PROGRAM PRG_HMIControl
VAR
//Motor 1 Animation
rM1MotorPosition     : LREAL;  // Real Motor Actual position
rM1MotorPositionPerc : LREAL;  // Motor Actual Position Scaled 0-100
cM1MinPosition       : LREAL := 0.0; // Minimum expected Value
cM1MaxPosition       : LREAL := -320.0; // Maximum expected Value (Default Value)

//Motor 2 Animation
rM2MotorPosition     : LREAL;  // Real Motor Actual position
rM2MotorPositionPerc : LREAL;  // Motor Actual Position Scaled 0-100
cM2MinPosition       : LREAL := 0.0; // Minimum expected Value
cM2MaxPosition       : LREAL := -170.0; // Maximum expected Value (Default Value)

//Pumps Animation and status
aPumpStatus			: ARRAY[1..10] OF ST_ActuatorStatus;
fbBlinkPumpArrowFWD	: ARRAY[1..10] OF FB_Blink;
fbBlinkPumpArrowBWD	: ARRAY[1..10] OF FB_Blink;

//Headbar Machine Mode transition
fbBlinkMachineModeName 	: FB_Blink;
ePrevMode               : E_MachineMode := E_MachineMode.IMEDIATE_FAULT; 
rTrigChange             : R_TRIG;
bStateChanged           : BOOL;
tpChangePulse           : TP; // gera um pulso de PT quando IN sobe
bBlinkMode              : BOOL;

//Doors Animation
fbBlinkDoor	: ARRAY[1..6] OF FB_Blink;
fbHMIScan	: FB_Blink;

//Icons Animation
bFirstIconSet : BOOL := FALSE;

//EStops Buttons
fbBlinkEStopSide	: FB_Blink;
fbBlinkEStopFront	: FB_Blink;

//Solvent status flags
bSolventIssue : BOOL := FALSE;
ton500ms : TON;
i : INT;

//Timers for releasing interlock signals.
tonInterlockReleaseM1 : ton;
tonInterlockReleaseM2 : ton;
tonInterlockReleaseM3 : ton;

//Jars Animation
curTurns         : LREAL;
deltaTurns       : LREAL;
dMl              : LREAL;
dir              : SINT;       // -1 Fill down, +1 Fill up, 0 stopped
effDeltaMl       : LREAL;
valIdx           : INT;
displayMl        : LREAL;
segPrevEff       : LREAL;
segNowEff        : LREAL;
bRecircActive    : BOOL;
END_VAR

VAR CONSTANT
    cJarsCount              : INT   := 10;
    cJarCapacity_ml         : LREAL := 80.0;
    cDeadVolDefault_ml      : LREAL := 20.0;
    cEpsTurns               : LREAL := 1e-6;
    cRecircLowDeg           : LREAL := 4700.0;
    cRecircHighDeg          : LREAL := 4900.0;
    cRecircDisplayMin_ml    : LREAL := 20.0;   // alvo mínimo visual durante recirculação
END_VAR

VAR RETAIN
    // Integração por bomba (estado interno do jar)
    aPrevTurns       : ARRAY[1..10] OF LREAL;
    aPrevInit        : ARRAY[1..10] OF BOOL;
    aJarMl           : ARRAY[1..10] OF LREAL;

    // Segmentação por direção (fora da recirculação)
    aSegDir          : ARRAY[1..10] OF SINT;     // -1 / 0 / +1
    aSegAbsMl        : ARRAY[1..10] OF LREAL;    // mL acumulados no segmento atual (|mL|)
    aSegAbsMlPrev    : ARRAY[1..10] OF LREAL;

    // Ajustes de unidade e dead volume por bomba
    aUnitsPerTurn    : ARRAY[1..10] OF LREAL := [1(360.0),360.0,360.0,360.0,360.0,360.0,360.0,360.0,360.0,360.0]; // graus->volta
    aDeadVolCfg_ml   : ARRAY[1..10] OF LREAL := [1(cDeadVolDefault_ml),
                                                 cDeadVolDefault_ml, cDeadVolDefault_ml, cDeadVolDefault_ml, cDeadVolDefault_ml,
                                                 cDeadVolDefault_ml, cDeadVolDefault_ml, cDeadVolDefault_ml, cDeadVolDefault_ml, cDeadVolDefault_ml];

    // Exibição durante recirculação
    aRecircWasActive : ARRAY[1..10] OF BOOL;     // para detectar borda de entrada/saída
    aRecircBaseMl    : ARRAY[1..10] OF LREAL;    // patamar antes de entrar em recirculação
    aDispMl          : ARRAY[1..10] OF LREAL;    // nível exibido (pode divergir de aJarMl na recirculação)
END_VAR

//Buttons Indicators -------------------------------------------------------------------------------------------------
GVL_HMI.HMIDigOutputs.bHMIResetButton 	:= GVL_IO.gDigOutputs.bResetIndicator;
GVL_HMI.HMIDigOutputs.bHMIStartButton	:= GVL_IO.gDigOutputs.bStartIndicator;
fbBlinkEStopSide(bEnable := NOT (GVL_Safety.SafetyInputs.bEStopSideCh1 OR GVL_Safety.SafetyInputs.bEStopSideCh2), tPeriod := T#1S); //EStop Button located on side Flashing FB
fbBlinkEStopFront(bEnable := NOT (GVL_Safety.SafetyInputs.bEStopHMICh1 OR GVL_Safety.SafetyInputs.bEStopHMICh2), tPeriod := T#1S);  //EStop Button located on front Flashing FB
GVL_HMI.HMIDigOutputs.bHMIEStopSide		:= fbBlinkEStopSide.bBlink;
GVL_HMI.HMIDigOutputs.bHMIEStopFront	:= fbBlinkEStopFront.bBlink;

(* Alarm Lamp Indicator for HMI --------------------------------------------------------------------------------------- *)
GVL_HMI.HMIDigOutputs.bAlarmLampRed 	:= GVL_IO.gDigOutputs.bTowerRedLight; 	//Red Light
GVL_HMI.HMIDigOutputs.bAlarmLampAmbar 	:= GVL_IO.gDigOutputs.bTowerAmberLight; //Ambar Light
GVL_HMI.HMIDigOutputs.bAlarmLampGreen 	:= GVL_IO.gDigOutputs.bTowerGreenLight; //Green Light

(* <Controls Animation> ------------------------------------------------------------------------------------------------ *)
ACT_M1Animation();
ACT_M2Animation();

(* Head Bar Blinking *) //----------------------------------------------------------------------------------------------------
// 1) State changed?
rTrigChange(CLK := (GVL_HMI.eMachineMode <> ePrevMode));
bStateChanged := rTrigChange.Q;

// 2) Short pulse whe changed
tpChangePulse(IN := bStateChanged, PT := T#500MS);

// 3) Blinking states
bBlinkMode := (GVL_HMI.eMachineMode = E_MachineMode.SYSTEM_READY)
           OR (GVL_HMI.eMachineMode = E_MachineMode.IMEDIATE_FAULT);

// Blinking F
fbBlinkMachineModeName(bEnable := bBlinkMode, tPeriod := T#1S);

// 4) HMI Output
GVL_HMI.bMachineModeBlinking := tpChangePulse.Q OR (bBlinkMode AND fbBlinkMachineModeName.bBlink);

// 5) Update previous machine mode
ePrevMode := GVL_HMI.eMachineMode;

(* HMI Lights Control *) //-----------------------------------------------------------------------------------------------
GVL_IO.gRelayOutputs.bSampleRecoveryLight 		:= GVL_HMI.bLightsToggleButton;
GVL_IO.gRelayOutputs.bStageCollectionLeftLight 	:= GVL_HMI.bLightsToggleButton;
GVL_IO.gRelayOutputs.bStageCollectionRightLight := GVL_HMI.bLightsToggleButton;

(* <Linear Pumps Old Position> ----------------------------------------------------------------------------------------- *)
// display linear pumps old position saved on persistent memory when in Calibration Mode
IF GVL_HMI.eMachineMode = E_MachineMode.CALIBRATION THEN
	FOR i := 1 TO 10 DO
		GVL_HMI.aCalibLinearPumps[i].rOldPosition := GVL_Retain.rLinearPumpOldPosition[i];
		//pump factor
		GVL_HMI.aCalibLinearPumps[i].rPumpFactor := GVL_Motion.aPumps[1].Rotary.rActualPos;
	END_FOR
END_IF

(* <Pump Factor Showing> ----------------------------------------------------------------------------------------------- *)
(*IF GVL_HMI.eMachineMode = E_MachineMode.CALIBRATION THEN
	FOR i := 1 TO 10 DO
		GVL_HMI.aCalPumpResults[i].rPumpFactor := GVL_Motion.aPumps[i].Rotary.rPumpFactorFromCalBox;
	END_FOR
END_IF
*)

(* <Safety Controls> ----------------------------------------------------------------------------------------------------*)
ton500ms(IN := NOT ton500ms.Q, PT := T#500MS);

IF ton500ms.Q THEN ACT_IOControls(); END_IF

//Calibration Box presence
GVL_HMI.bHMICalibrationBox := GVL_IO.gDigInputs.bCalibrationBoxPresent;

//Valves Angle
GVL_HMI.HMIAnimation.aValveAngle[1]	:= GVL_Motion.aValves[1].rActualPosition / 60;
GVL_HMI.HMIAnimation.aValveAngle[2]	:= GVL_Motion.aValves[2].rActualPosition / 60;;
GVL_HMI.HMIAnimation.aValveAngle[3]	:= GVL_Motion.aValves[3].rActualPosition / 60;;
GVL_HMI.HMIAnimation.aValveAngle[4]	:= GVL_Motion.aValves[4].rActualPosition / 60;;
GVL_HMI.HMIAnimation.aValveAngle[5]	:= GVL_Motion.aValves[5].rActualPosition / 60;;

//Pumps status Running or busy
IF GVL_HMI.eMachineMode = E_MachineMode.MANUAL THEN
	FOR i := 1 TO 10 DO
		aPumpStatus[i] := GVL_Motion.aPumpsRotary[i].GetStatus();
		GVL_HMI.aManualPumpsCmd[i].bBusy := NOT GVL_Motion.aPumps[i].Rotary.iNotMoving; //aPumpStatus[i].bBusy;
	END_FOR
END_IF

//Check if there is at least one pump running
GVL_Motion.bAnyPumpRunning := FALSE;
FOR i := 1 TO 10 DO
	IF GVL_HMI.aManualPumpsCmd[i].bBusy THEN
		GVL_Motion.bAnyPumpRunning := TRUE;
		EXIT;
	END_IF
END_FOR


//Pumps Animation | Calibration Screen
IF GVL_HMI.eMachineMode = E_MachineMode.CALIBRATION THEN
	ACT_CalibrationArrows();
END_IF

//Scan period for hmi refresh
//IF GVL_HMI.eMachineMode <> E_MachineMode.CALIBRATION AND GVL_HMI.eMachineMode <> E_MachineMode.MANUAL THEN
	fbHMIScan(bEnable := GVL_HMI.bHomeScreenLoaded, tPeriod := T#500MS);
	GVL_HMI.bMachineModeScan := fbHMIScan.bBlink;
//ELSE
//	GVL_HMI.bMachineModeScan := FALSE;
//END_IF


//Doors hide/visible 
GVL_HMI.HMIAnimation.bHMIDoorOpen[1] := NOT GVL_Safety.SafetyInputs.bStageCollectLeftDoorFdbk;
GVL_HMI.HMIAnimation.bHMIDoorOpen[2] := NOT GVL_Safety.SafetyInputs.bStageCollectRightDoorFdbk;
GVL_HMI.HMIAnimation.bHMIDoorOpen[3] := NOT GVL_Safety.SafetyInputs.bSampleRecoveryDoorFdbk;
GVL_HMI.HMIAnimation.bHMIDoorOpen[4] := GVL_IO.gDigInputs.bAccessDoor4InterlockFdbk;
GVL_HMI.HMIAnimation.bHMIDoorOpen[5] := GVL_IO.gDigInputs.bAccessDoor5InterlockFdbk;
GVL_HMI.HMIAnimation.bHMIDoorOpen[6] := GVL_IO.gDigInputs.bAccessDoor6InterlockFdbk;

//Doors open blinking red alert
fbBlinkDoor[1](bEnable := NOT GVL_Safety.SafetyInputs.bStageCollectLeftDoorFdbk, tPeriod := T#1S);
GVL_HMI.HMIAnimation.bHMIDoorBlink[1] := fbBlinkDoor[1].bBlink;

fbBlinkDoor[2](bEnable := NOT GVL_Safety.SafetyInputs.bStageCollectRightDoorFdbk, tPeriod := T#1S);
GVL_HMI.HMIAnimation.bHMIDoorBlink[2] := fbBlinkDoor[2].bBlink;

fbBlinkDoor[3](bEnable := NOT GVL_Safety.SafetyInputs.bSampleRecoveryDoorFdbk, tPeriod := T#1S);
GVL_HMI.HMIAnimation.bHMIDoorBlink[3] := fbBlinkDoor[3].bBlink;

fbBlinkDoor[4](bEnable := GVL_IO.gDigInputs.bAccessDoor4InterlockFdbk, tPeriod := T#1S);
GVL_HMI.HMIAnimation.bHMIDoorBlink[4] := fbBlinkDoor[4].bBlink;

fbBlinkDoor[5](bEnable := GVL_IO.gDigInputs.bAccessDoor5InterlockFdbk, tPeriod := T#1S);
GVL_HMI.HMIAnimation.bHMIDoorBlink[5] := fbBlinkDoor[5].bBlink;

fbBlinkDoor[6](bEnable := GVL_IO.gDigInputs.bAccessDoor6InterlockFdbk, tPeriod := T#1S);
GVL_HMI.HMIAnimation.bHMIDoorBlink[6] := fbBlinkDoor[6].bBlink;


(* <\Controls Animation> *********************************************************************************************** *)

(* <Icons Animation> *************************************************************************************************** *)
IF NOT bFirstIconSet THEN
	GVL_HMI.HMIAnimation.eIconStateSafety   := E_IconState.Waiting;
	GVL_HMI.HMIAnimation.eIconStateAirFlow  := E_IconState.Waiting;
	GVL_HMI.HMIAnimation.eIconStateHardware := E_IconState.Waiting;
	GVL_HMI.HMIAnimation.eIconStateLeakTest := E_IconState.Waiting;
	GVL_HMI.HMIAnimation.eIconStateRecovery := E_IconState.Waiting;
	GVL_HMI.HMIAnimation.eIconStateWashing  := E_IconState.Waiting;
	GVL_HMI.HMIAnimation.eIconStateDry 		:= E_IconState.Waiting;
	bFirstIconSet := TRUE;
END_IF

IF GVL_HMI.eMachineMode = E_MachineMode.IMEDIATE_FAULT THEN
	GVL_HMI.HMIAnimation.eIconStateSafety   := E_IconState.Waiting;
	GVL_HMI.HMIAnimation.eIconStateAirFlow  := E_IconState.Waiting;
	GVL_HMI.HMIAnimation.eIconStateHardware := E_IconState.Waiting;
	GVL_HMI.HMIAnimation.eIconStateLeakTest := E_IconState.Waiting;
	GVL_HMI.HMIAnimation.eIconStateRecovery := E_IconState.Waiting;
	GVL_HMI.HMIAnimation.eIconStateWashing  := E_IconState.Waiting;
	GVL_HMI.HMIAnimation.eIconStateDry 	    := E_IconState.Waiting;
ELSE
	GVL_HMI.HMIAnimation.eIconStateSafety := E_IconState.Completed;
END_IF

IF GVL_HMI.eMachineMode = E_MachineMode.STOPPED THEN
	GVL_HMI.HMIAnimation.eIconStateSafety   := E_IconState.Waiting;
	GVL_HMI.HMIAnimation.eIconStateAirFlow  := E_IconState.Waiting;
	GVL_HMI.HMIAnimation.eIconStateHardware := E_IconState.Waiting;
	GVL_HMI.HMIAnimation.eIconStateLeakTest := E_IconState.Waiting;
	GVL_HMI.HMIAnimation.eIconStateRecovery := E_IconState.Waiting;
	GVL_HMI.HMIAnimation.eIconStateWashing  := E_IconState.Waiting;
	GVL_HMI.HMIAnimation.eIconStateDry 	    := E_IconState.Waiting;
END_IF

(* <\Icons Animation> *************************************************************************************************** *)

(* <Machine Settings> ************************************************************************************************** *)
IF GVL_HMI.bSaveParametersBt THEN // Save Settings button from HMI
	GVL_Settings.stMachineParam	 		:= GVL_HMI.HMIParameters; 		 // Motion Settings
	GVL_Settings.stCalibParameters 		:= GVL_HMI.stHMICalibParameters; // Calibration Settings
	GVL_Settings.stPumpParameters 		:= GVL_HMI.stHMIPumpParameters;	 // Pump Settings
	GVL_Settings.stLeakTestParameters 	:= GVL_HMI.stLeakTestParameters; // Leak Test Settings
	GVL_HMI.bSaveParametersBt 	:= FALSE;
	GVL_HMI.bSaveParametersDone := TRUE;
END_IF

IF GVL_HMI.bReloadHMIParameters OR (GVL_HMI.eMachineMode = E_MachineMode.CALIBRATION) THEN
	GVL_HMI.HMIParameters := GVL_Settings.stMachineParam;				 // Motion Settings
	GVL_HMI.stHMICalibParameters := GVL_Settings.stCalibParameters; 	 // Calibration Settings
	GVL_HMI.stHMIPumpParameters  := GVL_Settings.stPumpParameters; 		 // Pump Settings
	GVL_HMI.stLeakTestParameters := GVL_Settings.stLeakTestParameters; 	 // Leak Test Settings
	GVL_HMI.bReloadHMIParameters := FALSE;
END_IF
(* <\Machine Settings> ************************************************************************************************** *)

(* <HMI Alerts> ********************************************************************************************************* *)

//Auto Cycle Incoherence [when there is something missing to start the auto cycle] 
GVL_HMI.bIncoherenceDetected := (NOT GVL_Recipe.bIsThereRecipeActivated) OR (NOT GVL_IO.gDigInputs.bThroatJigPresent) OR (NOT GVL_IO.bVialRackPresent) OR bSolventIssue;

bSolventIssue := GVL_Alarms.aSolventLowLevel[1] OR GVL_Alarms.aSolventLowLevel[2] OR GVL_Alarms.aSolventLowLevel[3] OR GVL_Alarms.aSolventLowLevel[4] OR GVL_Alarms.bWasteHighLevel;

IF GVL_HMI.HMIAnimation.rWasteLevel	> 70 THEN
	GVL_Alarms.bWasteHighLevel := TRUE;
ELSE
	GVL_Alarms.bWasteHighLevel := FALSE;
END_IF

IF GVL_Recipe.bIsThereRecipeActivated THEN
	//Checking solvent levels of Rinse 1 Solvent
	CASE GVL_Recipe.stActiveRecipe.stSolventsTimes.aSolventN[1] OF
	1:
		IF GVL_HMI.HMIAnimation.aSolventLevel[1] < 30 THEN
			GVL_Alarms.aSolventLowLevel[1] := TRUE;
		ELSE
			GVL_Alarms.aSolventLowLevel[1] := FALSE;
		END_IF
	2:
		IF GVL_HMI.HMIAnimation.aSolventLevel[2] < 30 THEN
			GVL_Alarms.aSolventLowLevel[2] := TRUE;
		ELSE
			GVL_Alarms.aSolventLowLevel[2] := FALSE;
		END_IF

	3:
		IF GVL_HMI.HMIAnimation.aSolventLevel[3] < 30 THEN
			GVL_Alarms.aSolventLowLevel[3] := TRUE;
		ELSE
			GVL_Alarms.aSolventLowLevel[3] := FALSE;
		END_IF
	4:
		IF GVL_HMI.HMIAnimation.aSolventLevel[4] < 30 THEN
			GVL_Alarms.aSolventLowLevel[4] := TRUE;
		ELSE
			GVL_Alarms.aSolventLowLevel[4] := FALSE;
		END_IF
	END_CASE 
	
	//Checking solvent levels of Rinse 2 Solvent
	CASE GVL_Recipe.stActiveRecipe.stSolventsTimes.aSolventN[2] OF
	1:
		IF GVL_HMI.HMIAnimation.aSolventLevel[1] < 30 THEN
			GVL_Alarms.aSolventLowLevel[1] := TRUE;
		ELSE
			GVL_Alarms.aSolventLowLevel[1] := FALSE;
		END_IF
	2:
		IF GVL_HMI.HMIAnimation.aSolventLevel[2] < 30 THEN
			GVL_Alarms.aSolventLowLevel[2] := TRUE;
		ELSE
			GVL_Alarms.aSolventLowLevel[2] := FALSE;
		END_IF

	3:
		IF GVL_HMI.HMIAnimation.aSolventLevel[3] < 30 THEN
			GVL_Alarms.aSolventLowLevel[3] := TRUE;
		ELSE
			GVL_Alarms.aSolventLowLevel[3] := FALSE;
		END_IF
	4:
		IF GVL_HMI.HMIAnimation.aSolventLevel[4] < 30 THEN
			GVL_Alarms.aSolventLowLevel[4] := TRUE;
		ELSE
			GVL_Alarms.aSolventLowLevel[4] := FALSE;
		END_IF
	END_CASE 
END_IF

//-------------------------------------------------

IF GVL_Recipe.bIsThereRecipeActivated THEN
	GVL_HMI.sActivatedRecipeHomeNaming := concat(GVL_Recipe.stActiveRecipe.stInfo.sMethodName,concat(' | Created by ', concat(GVL_Recipe.stActiveRecipe.stInfo.sCreatedBy,concat(' on ', DATE_TO_STRING(GVL_Recipe.stActiveRecipe.stInfo.dCreationDate)))));
ELSE
	GVL_HMI.sActivatedRecipeHomeNaming := 'There is no Recipe Activated';
END_IF

(* <\HMI Alerts> ******************************************************************************************************* *)
(* Motors Interlock *) // Releasing alarm trigger after 2 seconds.
IF GVL_HMI.bM1MoveNotAllowedTrigger THEN
	tonInterlockReleaseM1(In := TRUE, PT := T#2S);
ELSE
	tonInterlockReleaseM1(In := FALSE, PT := T#2S);
END_IF

IF GVL_HMI.bM2MoveNotAllowedTrigger THEN
	tonInterlockReleaseM2(In := TRUE, PT := T#2S);
ELSE
	tonInterlockReleaseM2(In := FALSE, PT := T#2S);
END_IF

IF GVL_HMI.bM3MoveNotAllowedTrigger THEN
	tonInterlockReleaseM3(In := TRUE, PT := T#2S);
ELSE
	tonInterlockReleaseM3(In := FALSE, PT := T#2S);
END_IF

IF tonInterlockReleaseM1.Q THEN
	GVL_HMI.bM1MoveNotAllowedTrigger := FALSE;
END_IF

IF tonInterlockReleaseM2.Q THEN
	GVL_HMI.bM2MoveNotAllowedTrigger := FALSE;
END_IF

IF tonInterlockReleaseM3.Q THEN
	GVL_HMI.bM3MoveNotAllowedTrigger := FALSE;
END_IF

(* <TEMP ******************************************************************************************************* *)
IF GVL_HMI.bResetM1MotorBt THEN
	GVL_HMI.bResetM1MotorBt := NOT GVL_Motion.aMotors[1].Reset();
END_IF

ACTION ACT_CalibrationArrows:
(* Pumps arrow animation *)
//Get pump Status
FOR i := 1 TO 10 DO
	aPumpStatus[i] := GVL_Motion.aPumpsRotary[i].GetStatus();
END_FOR

//Blink aPumpMovingFwd[i] if moving forward
FOR i := 1 TO 10 DO
	fbBlinkPumpArrowFWD[i]( bEnable := aPumpStatus[i].bMovingFwd, tPeriod := T#500MS );
	GVL_HMI.HMIAnimation.aPumpingArrowFwd[i] := fbBlinkPumpArrowFWD[i].bBlink;
END_FOR

//Blink aPumpMovingBwd[i] if moving backwards
FOR i := 1 TO 10 DO
	fbBlinkPumpArrowBWD[i]( bEnable := aPumpStatus[i].bMovingBck, tPeriod := T#500MS );
	GVL_HMI.HMIAnimation.aPumpingArrowBwd[i] := fbBlinkPumpArrowBWD[i].bBlink;
END_FOR
END_ACTION

ACTION ACT_IOControls:

(* <EL6910 Terminal 3> -------------------------------------------------------------------------------------------------------------*)
GVL_IO.stEL6910.qSafetyRun 			:= GVL_Safety.bSafetyRun;
GVL_IO.stEL6910.qSafetyErrorAck 	:= GVL_Safety.bSafetyErrorAck;
GVL_IO.stEL6910.qSafetyAirPresureOK := GVL_Safety.SafetyOutputs.bAirPressureOK;
GVL_IO.stEL6910.iSafetyOK 			:= GVL_Safety.bSafetyEnable;
GVL_IO.stEL6910.qLockDoorsCommand	:= GVL_Safety.bDoorLockCommand;
GVL_IO.stEL6910.iBypassDoor3Command := GVL_Safety.bDoor3BypassAccepted;


(* <EL1918 Terminal 4> -------------------------------------------------------------------------------------------------------------*)
GVL_HMI.aIOTerm04[1] := GVL_Safety.SafetyInputs.bEStopHMICh1;
GVL_HMI.aIOTerm04[2] := GVL_Safety.SafetyInputs.bEStopHMICh2;
GVL_HMI.aIOTerm04[3] := GVL_Safety.SafetyInputs.bEStopSideCh1;
GVL_HMI.aIOTerm04[4] := GVL_Safety.SafetyInputs.bEStopSideCh2;
GVL_HMI.aIOTerm04[5] := GVL_Safety.SafetyInputs.bMachineReset;
GVL_HMI.aIOTerm04[6] := GVL_Safety.SafetyInputs.bStageCollectLeftDoorCh1;
GVL_HMI.aIOTerm04[7] := GVL_Safety.SafetyInputs.bStageCollectLeftDoorCh2;
GVL_HMI.aIOTerm04[8] := GVL_Safety.SafetyInputs.bStageCollectLeftDoorFdbk;

(* <EL1918 Terminal 5> -------------------------------------------------------------------------------------------------------------*)
GVL_HMI.aIOTerm05[1] := GVL_Safety.SafetyInputs.bStageCollectRightDoorCh1;
GVL_HMI.aIOTerm05[2] := GVL_Safety.SafetyInputs.bStageCollectRightDoorCh2;
GVL_HMI.aIOTerm05[3] := GVL_Safety.SafetyInputs.bStageCollectRightDoorFdbk;
GVL_HMI.aIOTerm05[4] := GVL_Safety.SafetyInputs.bSampleRecoveryDoorCh1;
GVL_HMI.aIOTerm05[5] := GVL_Safety.SafetyInputs.bSampleRecoveryDoorCh2;
GVL_HMI.aIOTerm05[6] := GVL_Safety.SafetyInputs.bSampleRecoveryDoorFdbk;
GVL_HMI.aIOTerm05[7] := FALSE;
GVL_HMI.aIOTerm05[8] := FALSE;

(* <EL1918 Terminal 6> -------------------------------------------------------------------------------------------------------------*)
GVL_HMI.aIOTerm06[1] := NOT GVL_Safety.SafetyInputs.bFestoMS6ValveFdbk;
GVL_HMI.aIOTerm06[2] := GVL_Safety.SafetyInputs.bFestoMS6DumpValveFdbk;
GVL_HMI.aIOTerm06[3] := NOT GVL_Safety.SafetyInputs.bD4AccessDoorIntlckOSSD1;
GVL_HMI.aIOTerm06[4] := NOT GVL_Safety.SafetyInputs.bD4AccessDoorIntlckOSSD2;
GVL_HMI.aIOTerm06[5] := NOT GVL_Safety.SafetyInputs.bD5AccessDoorIntlckOSSD1;
GVL_HMI.aIOTerm06[6] := NOT GVL_Safety.SafetyInputs.bD5AccessDoorIntlckOSSD2;
GVL_HMI.aIOTerm06[7] := NOT GVL_Safety.SafetyInputs.bD6AccessDoorIntlckOSSD1;
GVL_HMI.aIOTerm06[8] := NOT GVL_Safety.SafetyInputs.bD6AccessDoorIntlckOSSD2;

(* <EL2904 Terminal 7> -------------------------------------------------------------------------------------------------------------*)
GVL_HMI.aIOTerm07[1] := GVL_Safety.aEL2904_T07[1];
GVL_HMI.aIOTerm07[2] := GVL_Safety.aEL2904_T07[2];
GVL_HMI.aIOTerm07[3] := GVL_Safety.aEL2904_T07[3];
GVL_HMI.aIOTerm07[4] := GVL_Safety.aEL2904_T07[4];

(* <EL2904 Terminal 8> -------------------------------------------------------------------------------------------------------------*)
GVL_HMI.aIOTerm08[1] := GVL_Safety.aEL2904_T08[1];
GVL_HMI.aIOTerm08[2] := GVL_Safety.aEL2904_T08[2];
GVL_HMI.aIOTerm08[3] := GVL_Safety.aEL2904_T08[3];
GVL_HMI.aIOTerm08[4] := GVL_Safety.aEL2904_T08[4];

(* <EL1809 Terminal 9> -------------------------------------------------------------------------------------------------------------*)
GVL_HMI.aIOTerm09[1] := GVL_IO.gDigInputs.bStartButton;
GVL_HMI.aIOTerm09[2] := GVL_IO.gDigInputs.bStopButton;
GVL_HMI.aIOTerm09[3] := GVL_IO.gDigInputs.b24VPowerSupplyOK;
GVL_HMI.aIOTerm09[4] := GVL_IO.gDigInputs.b24VPowerSupplyOKBck;
GVL_HMI.aIOTerm09[5] := GVL_IO.gDigInputs.b48VPowerSupplyOK;
GVL_HMI.aIOTerm09[6] := GVL_IO.gDigInputs.bStageCollection_Home;
GVL_HMI.aIOTerm09[7] := GVL_IO.gDigInputs.bSampleRecovery_Vertical_Home;
GVL_HMI.aIOTerm09[8] := GVL_IO.gDigInputs.bSampleRecovery_Horizontal_Home;
GVL_HMI.aIOTerm09[9] := GVL_IO.gDigInputs.bWasteOverflowSensor;
GVL_HMI.aIOTerm09[10] := GVL_IO.gDigInputs.bUPSReady;
GVL_HMI.aIOTerm09[11] := GVL_IO.gDigInputs.bUPSReplaceBattery;
GVL_HMI.aIOTerm09[12] := GVL_IO.gDigInputs.b48VPowerSupplyOKBck;
GVL_HMI.aIOTerm09[13] := GVL_IO.gDigInputs.bCalibrationBoxPresent;
GVL_HMI.aIOTerm09[14] := GVL_IO.gDigInputs.bThroatJigPresent;
GVL_HMI.aIOTerm09[15] := FALSE;
GVL_HMI.aIOTerm09[16] := FALSE;

(* <EL2809 Terminal 10> -------------------------------------------------------------------------------------------------------------*)
GVL_HMI.aIOTerm10[1] := GVL_IO.gDigOutputs.bStartIndicator;
GVL_HMI.aIOTerm10[2] := GVL_IO.gDigOutputs.bResetIndicator;
GVL_HMI.aIOTerm10[3] := GVL_IO.gDigOutputs.bTowerRedLight;
GVL_HMI.aIOTerm10[4] := GVL_IO.gDigOutputs.bTowerAmberLight;
GVL_HMI.aIOTerm10[5] := GVL_IO.gDigOutputs.bTowerGreenLight;
GVL_HMI.aIOTerm10[6] := GVL_IO.gDigOutputs.bTowerBuzzer;
GVL_HMI.aIOTerm10[7] := GVL_IO.gDigOutputs.bSolenoidValveB;
GVL_HMI.aIOTerm10[8] := GVL_IO.gDigOutputs.bSolenoidValveA;
GVL_HMI.aIOTerm10[9] := GVL_IO.gDigOutputs.bSolenoidValveC;
GVL_HMI.aIOTerm10[10] := FALSE;
GVL_HMI.aIOTerm10[11] := FALSE;
GVL_HMI.aIOTerm10[12] := FALSE;
GVL_HMI.aIOTerm10[13] := FALSE;
GVL_HMI.aIOTerm10[14] := FALSE;
GVL_HMI.aIOTerm10[15] := FALSE;
GVL_HMI.aIOTerm10[16] := FALSE;

(* <EL2624 Terminal 11> -------------------------------------------------------------------------------------------------------------*)
GVL_HMI.aIOTerm11[1] := GVL_IO.gRelayOutputs.bStageCollectionLeftLight;
GVL_HMI.aIOTerm11[2] := GVL_IO.gRelayOutputs.bSampleRecoveryLight;
GVL_HMI.aIOTerm11[3] := GVL_IO.gRelayOutputs.bStageCollectionRightLight;
GVL_HMI.aIOTerm11[4] := FALSE;

(* <EL9410 Terminal 12> -------------------------------------------------------------------------------------------------------------*)
GVL_HMI.aIOTerm12[1] := GVL_IO.bEL9410UPStatus;
GVL_HMI.aIOTerm12[2] := GVL_IO.bEL9410USStatus;

(* <EL3058 Terminal 13> -------------------------------------------------------------------------------------------------------------*)
GVL_HMI.aIOTerm13[1] := GVL_IO.gAnalogInputs.rMainPressureSupplyInput;
GVL_HMI.aIOTerm13[2] := GVL_IO.gAnalogInputs.rLeakTestPressureSensor;
GVL_HMI.aIOTerm13[3] := GVL_IO.gAnalogInputs.rPressureRegulatorInput;
GVL_HMI.aIOTerm13[3] := 0.0;

(* <EL9576 Terminal 14> -------------------------------------------------------------------------------------------------------------*)
GVL_HMI.aIOTerm14[1] := GVL_IO.bEL9576T14Overtemp;
GVL_HMI.aIOTerm14[2] := GVL_IO.bEL9576T14I2TError;
GVL_HMI.aIOTerm14[3] := GVL_IO.bEL9576T14I2TWarning;
GVL_HMI.aIOTerm14[4] := GVL_IO.bEL9576T14OverVoltage;
GVL_HMI.aIOTerm14[5] := GVL_IO.bEL9576T14UnderVoltage;
GVL_HMI.aIOTerm14[6] := GVL_IO.bEL9576T14ChopperOn;
GVL_HMI.aIOTerm14[7] := GVL_IO.bEL9576T14OverCurrent;
GVL_HMI.iIOTerm14DCIn := GVL_IO.bEL9576T14DCLinkVoltage;

(* <EL7211 Terminal 15> -------------------------------------------------------------------------------------------------------------*)
GVL_HMI.aIOTerm15[1] := GVL_Motion.M2Motor.iOperational;
GVL_HMI.aIOTerm15[2] := GVL_Motion.M2Motor.iHomed;
GVL_HMI.aIOTerm15[3] := GVL_Motion.M2Motor.iError;
GVL_HMI.aIOTerm15Values[1] := LINT_TO_LREAL(TRUNC(GVL_Motion.M2Motor.rActualPosition*1000)) / 1000.0;
GVL_HMI.aIOTerm15Values[2] := LINT_TO_LREAL(TRUNC(GVL_Motion.M2Motor.rActualVel*1000)) / 1000.0;
GVL_HMI.aIOTerm15Values[3] := LINT_TO_LREAL(TRUNC(GVL_Motion.M2Motor.rActualTorque*1000)) / 1000.0;
GVL_HMI.iIOTerm15ErrorCode := GVL_Motion.M2Motor.nErrorCode;

(* <EL7211 Terminal 16> -------------------------------------------------------------------------------------------------------------*)
GVL_HMI.aIOTerm16[1] := GVL_Motion.M3Motor.iOperational;
GVL_HMI.aIOTerm16[2] := GVL_Motion.M3Motor.iHomed;
GVL_HMI.aIOTerm16[3] := GVL_Motion.M3Motor.iError;
GVL_HMI.aIOTerm16Values[1] := LINT_TO_LREAL(TRUNC(GVL_Motion.M3Motor.rActualPosition*1000)) / 1000.0;
GVL_HMI.aIOTerm16Values[2] := LINT_TO_LREAL(TRUNC(GVL_Motion.M3Motor.rActualVel*1000)) / 1000.0;
GVL_HMI.aIOTerm16Values[3] := LINT_TO_LREAL(TRUNC(GVL_Motion.M3Motor.rActualTorque*1000)) / 1000.0;
GVL_HMI.iIOTerm16ErrorCode := GVL_Motion.M3Motor.nErrorCode;

(* <EL3022 Terminal 17> -------------------------------------------------------------------------------------------------------------*)
GVL_HMI.aIOTerm17[1] := GVL_IO.bEL3022ChAUnderRange;
GVL_HMI.aIOTerm17[2] := GVL_IO.bEL3022ChAOverRange;
GVL_HMI.aIOTerm17[3] := GVL_IO.bEL3022ChAError;
GVL_HMI.aIOTerm17[4] := GVL_IO.bEL3022ChBUnderRange;
GVL_HMI.aIOTerm17[5] := GVL_IO.bEL3022ChBOverRange;
GVL_HMI.aIOTerm17[6] := GVL_IO.bEL3022ChBError;
GVL_HMI.aIOTerm17Values[1] := 0.0;
GVL_HMI.aIOTerm17Values[2] := 0.0;

(* <EL1809 Terminal 18> -------------------------------------------------------------------------------------------------------------*)
GVL_HMI.aIOTerm18[1] := NOT GVL_IO.gDigInputs.bAccessDoor4InterlockFdbk;
GVL_HMI.aIOTerm18[2] := NOT GVL_IO.gDigInputs.bAccessDoor5InterlockFdbk;
GVL_HMI.aIOTerm18[3] := NOT GVL_IO.gDigInputs.bAccessDoor6InterlockFdbk;
GVL_HMI.aIOTerm18[4] := FALSE;
GVL_HMI.aIOTerm18[5] := FALSE;
GVL_HMI.aIOTerm18[6] := FALSE;
GVL_HMI.aIOTerm18[7] := FALSE;
GVL_HMI.aIOTerm18[8] := FALSE;
GVL_HMI.aIOTerm18[9] := FALSE;
GVL_HMI.aIOTerm18[10] := FALSE;
GVL_HMI.aIOTerm18[11] := FALSE;
GVL_HMI.aIOTerm18[12] := FALSE;
GVL_HMI.aIOTerm18[13] := FALSE;
GVL_HMI.aIOTerm18[14] := FALSE;
GVL_HMI.aIOTerm18[15] := FALSE;
GVL_HMI.aIOTerm18[16] := FALSE;

(* <EL2904 Terminal 19> -------------------------------------------------------------------------------------------------------------*)
GVL_HMI.aIOTerm19[1] := GVL_Safety.aEL2904_T19[1];
GVL_HMI.aIOTerm19[2] := GVL_Safety.aEL2904_T19[2];
GVL_HMI.aIOTerm19[3] := GVL_Safety.aEL2904_T19[3];
GVL_HMI.aIOTerm19[4] := GVL_Safety.aEL2904_T19[4];

(* <EL7062 Terminal 23> -------------------------------------------------------------------------------------------------------------*)
GVL_HMI.stIOTerm23.bAxisOperational[1] 	:= GVL_Motion.aPumps[1].Linear.iOperational;
GVL_HMI.stIOTerm23.rActualPosition[1] 	:= GVL_Motion.aPumps[1].Linear.rActualPos;
GVL_HMI.stIOTerm23.rActualVelocity[1] 	:= GVL_Motion.aPumps[1].Linear.rActualVel;
GVL_HMI.stIOTerm23.rActualTorque[1] 	:= GVL_Motion.aPumps[1].Linear.rActualTorque;
GVL_HMI.stIOTerm23.bAxisHomed[1] 		:= GVL_Motion.aPumps[1].Linear.iHomed;
GVL_HMI.stIOTerm23.bAxisError[1] 		:= GVL_Motion.aPumps[1].Linear.iError;
GVL_HMI.stIOTerm23.nErrorCode[1] 		:= GVL_Motion.aPumps[1].Linear.nErrorCode;
GVL_HMI.stIOTerm23.bAxisOperational[2] 	:= GVL_Motion.aPumps[1].Rotary.iOperational;
GVL_HMI.stIOTerm23.rActualPosition[2] 	:= GVL_Motion.aPumps[1].Rotary.rActualPos;
GVL_HMI.stIOTerm23.rActualVelocity[2] 	:= GVL_Motion.aPumps[1].Rotary.rActualVel;
GVL_HMI.stIOTerm23.rActualTorque[2] 	:= GVL_Motion.aPumps[1].Rotary.rActualTorque;
GVL_HMI.stIOTerm23.bAxisHomed[2] 		:= GVL_Motion.aPumps[1].Rotary.iHomed;
GVL_HMI.stIOTerm23.bAxisError[2] 		:= GVL_Motion.aPumps[1].Rotary.iError;
GVL_HMI.stIOTerm23.nErrorCode[2] 		:= GVL_Motion.aPumps[1].Rotary.nErrorCode;

(* <EL7062 Terminal 24> -------------------------------------------------------------------------------------------------------------*)
GVL_HMI.stIOTerm24.bAxisOperational[1] 	:= GVL_Motion.aPumps[2].Linear.iOperational;
GVL_HMI.stIOTerm24.rActualPosition[1] 	:= GVL_Motion.aPumps[2].Linear.rActualPos;
GVL_HMI.stIOTerm24.rActualVelocity[1] 	:= GVL_Motion.aPumps[2].Linear.rActualVel;
GVL_HMI.stIOTerm24.rActualTorque[1] 	:= GVL_Motion.aPumps[2].Linear.rActualTorque;
GVL_HMI.stIOTerm24.bAxisHomed[1] 		:= GVL_Motion.aPumps[2].Linear.iHomed;
GVL_HMI.stIOTerm24.bAxisError[1] 		:= GVL_Motion.aPumps[2].Linear.iError;
GVL_HMI.stIOTerm24.nErrorCode[1] 		:= GVL_Motion.aPumps[2].Linear.nErrorCode;
GVL_HMI.stIOTerm24.bAxisOperational[2] 	:= GVL_Motion.aPumps[2].Rotary.iOperational;
GVL_HMI.stIOTerm24.rActualPosition[2] 	:= GVL_Motion.aPumps[2].Rotary.rActualPos;
GVL_HMI.stIOTerm24.rActualVelocity[2] 	:= GVL_Motion.aPumps[2].Rotary.rActualVel;
GVL_HMI.stIOTerm24.rActualTorque[2] 	:= GVL_Motion.aPumps[2].Rotary.rActualTorque;
GVL_HMI.stIOTerm24.bAxisHomed[2] 		:= GVL_Motion.aPumps[2].Rotary.iHomed;
GVL_HMI.stIOTerm24.bAxisError[2] 		:= GVL_Motion.aPumps[2].Rotary.iError;
GVL_HMI.stIOTerm24.nErrorCode[2] 		:= GVL_Motion.aPumps[2].Rotary.nErrorCode;

(* <EL7062 Terminal 25> -------------------------------------------------------------------------------------------------------------*)
GVL_HMI.stIOTerm25.bAxisOperational[1] 	:= GVL_Motion.aPumps[3].Linear.iOperational;
GVL_HMI.stIOTerm25.rActualPosition[1] 	:= GVL_Motion.aPumps[3].Linear.rActualPos;
GVL_HMI.stIOTerm25.rActualVelocity[1] 	:= GVL_Motion.aPumps[3].Linear.rActualVel;
GVL_HMI.stIOTerm25.rActualTorque[1] 	:= GVL_Motion.aPumps[3].Linear.rActualTorque;
GVL_HMI.stIOTerm25.bAxisHomed[1] 		:= GVL_Motion.aPumps[3].Linear.iHomed;
GVL_HMI.stIOTerm25.bAxisError[1] 		:= GVL_Motion.aPumps[3].Linear.iError;
GVL_HMI.stIOTerm25.nErrorCode[1] 		:= GVL_Motion.aPumps[3].Linear.nErrorCode;
GVL_HMI.stIOTerm25.bAxisOperational[2] 	:= GVL_Motion.aPumps[3].Rotary.iOperational;
GVL_HMI.stIOTerm25.rActualPosition[2] 	:= GVL_Motion.aPumps[3].Rotary.rActualPos;
GVL_HMI.stIOTerm25.rActualVelocity[2] 	:= GVL_Motion.aPumps[3].Rotary.rActualVel;
GVL_HMI.stIOTerm25.rActualTorque[2] 	:= GVL_Motion.aPumps[3].Rotary.rActualTorque;
GVL_HMI.stIOTerm25.bAxisHomed[2] 		:= GVL_Motion.aPumps[3].Rotary.iHomed;
GVL_HMI.stIOTerm25.bAxisError[2] 		:= GVL_Motion.aPumps[3].Rotary.iError;
GVL_HMI.stIOTerm25.nErrorCode[2] 		:= GVL_Motion.aPumps[3].Rotary.nErrorCode;

(* <EL7062 Terminal 26> -------------------------------------------------------------------------------------------------------------*)
GVL_HMI.stIOTerm26.bAxisOperational[1] 	:= GVL_Motion.aPumps[4].Linear.iOperational;
GVL_HMI.stIOTerm26.rActualPosition[1] 	:= GVL_Motion.aPumps[4].Linear.rActualPos;
GVL_HMI.stIOTerm26.rActualVelocity[1] 	:= GVL_Motion.aPumps[4].Linear.rActualVel;
GVL_HMI.stIOTerm26.rActualTorque[1] 	:= GVL_Motion.aPumps[4].Linear.rActualTorque;
GVL_HMI.stIOTerm26.bAxisHomed[1] 		:= GVL_Motion.aPumps[4].Linear.iHomed;
GVL_HMI.stIOTerm26.bAxisError[1] 		:= GVL_Motion.aPumps[4].Linear.iError;
GVL_HMI.stIOTerm26.nErrorCode[1] 		:= GVL_Motion.aPumps[4].Linear.nErrorCode;
GVL_HMI.stIOTerm26.bAxisOperational[2] 	:= GVL_Motion.aPumps[4].Rotary.iOperational;
GVL_HMI.stIOTerm26.rActualPosition[2] 	:= GVL_Motion.aPumps[4].Rotary.rActualPos;
GVL_HMI.stIOTerm26.rActualVelocity[2] 	:= GVL_Motion.aPumps[4].Rotary.rActualVel;
GVL_HMI.stIOTerm26.rActualTorque[2] 	:= GVL_Motion.aPumps[4].Rotary.rActualTorque;
GVL_HMI.stIOTerm26.bAxisHomed[2] 		:= GVL_Motion.aPumps[4].Rotary.iHomed;
GVL_HMI.stIOTerm26.bAxisError[2] 		:= GVL_Motion.aPumps[4].Rotary.iError;
GVL_HMI.stIOTerm26.nErrorCode[2] 		:= GVL_Motion.aPumps[4].Rotary.nErrorCode;

(* <EL7062 Terminal 27> -------------------------------------------------------------------------------------------------------------*)
GVL_HMI.stIOTerm27.bAxisOperational[1] 	:= GVL_Motion.aPumps[5].Linear.iOperational;
GVL_HMI.stIOTerm27.rActualPosition[1] 	:= GVL_Motion.aPumps[5].Linear.rActualPos;
GVL_HMI.stIOTerm27.rActualVelocity[1] 	:= GVL_Motion.aPumps[5].Linear.rActualVel;
GVL_HMI.stIOTerm27.rActualTorque[1] 	:= GVL_Motion.aPumps[5].Linear.rActualTorque;
GVL_HMI.stIOTerm27.bAxisHomed[1] 		:= GVL_Motion.aPumps[5].Linear.iHomed;
GVL_HMI.stIOTerm27.bAxisError[1] 		:= GVL_Motion.aPumps[5].Linear.iError;
GVL_HMI.stIOTerm27.nErrorCode[1] 		:= GVL_Motion.aPumps[5].Linear.nErrorCode;
GVL_HMI.stIOTerm27.bAxisOperational[2] 	:= GVL_Motion.aPumps[5].Rotary.iOperational;
GVL_HMI.stIOTerm27.rActualPosition[2] 	:= GVL_Motion.aPumps[5].Rotary.rActualPos;
GVL_HMI.stIOTerm27.rActualVelocity[2] 	:= GVL_Motion.aPumps[5].Rotary.rActualVel;
GVL_HMI.stIOTerm27.rActualTorque[2] 	:= GVL_Motion.aPumps[5].Rotary.rActualTorque;
GVL_HMI.stIOTerm27.bAxisHomed[2] 		:= GVL_Motion.aPumps[5].Rotary.iHomed;
GVL_HMI.stIOTerm27.bAxisError[2] 		:= GVL_Motion.aPumps[5].Rotary.iError;
GVL_HMI.stIOTerm27.nErrorCode[2] 		:= GVL_Motion.aPumps[5].Rotary.nErrorCode;

(* <EL7062 Terminal 28> -------------------------------------------------------------------------------------------------------------*)
GVL_HMI.stIOTerm28.bAxisOperational[1] 	:= GVL_Motion.aPumps[6].Linear.iOperational;
GVL_HMI.stIOTerm28.rActualPosition[1] 	:= GVL_Motion.aPumps[6].Linear.rActualPos;
GVL_HMI.stIOTerm28.rActualVelocity[1] 	:= GVL_Motion.aPumps[6].Linear.rActualVel;
GVL_HMI.stIOTerm28.rActualTorque[1] 	:= GVL_Motion.aPumps[6].Linear.rActualTorque;
GVL_HMI.stIOTerm28.bAxisHomed[1] 		:= GVL_Motion.aPumps[6].Linear.iHomed;
GVL_HMI.stIOTerm28.bAxisError[1] 		:= GVL_Motion.aPumps[6].Linear.iError;
GVL_HMI.stIOTerm28.nErrorCode[1] 		:= GVL_Motion.aPumps[6].Linear.nErrorCode;
GVL_HMI.stIOTerm28.bAxisOperational[2] 	:= GVL_Motion.aPumps[6].Rotary.iOperational;
GVL_HMI.stIOTerm28.rActualPosition[2] 	:= GVL_Motion.aPumps[6].Rotary.rActualPos;
GVL_HMI.stIOTerm28.rActualVelocity[2] 	:= GVL_Motion.aPumps[6].Rotary.rActualVel;
GVL_HMI.stIOTerm28.rActualTorque[2] 	:= GVL_Motion.aPumps[6].Rotary.rActualTorque;
GVL_HMI.stIOTerm28.bAxisHomed[2] 		:= GVL_Motion.aPumps[6].Rotary.iHomed;
GVL_HMI.stIOTerm28.bAxisError[2] 		:= GVL_Motion.aPumps[6].Rotary.iError;
GVL_HMI.stIOTerm28.nErrorCode[2] 		:= GVL_Motion.aPumps[6].Rotary.nErrorCode;

(* <EL7062 Terminal 29> -------------------------------------------------------------------------------------------------------------*)
GVL_HMI.stIOTerm29.bAxisOperational[1] 	:= GVL_Motion.aPumps[7].Linear.iOperational;
GVL_HMI.stIOTerm29.rActualPosition[1] 	:= GVL_Motion.aPumps[7].Linear.rActualPos;
GVL_HMI.stIOTerm29.rActualVelocity[1] 	:= GVL_Motion.aPumps[7].Linear.rActualVel;
GVL_HMI.stIOTerm29.rActualTorque[1] 	:= GVL_Motion.aPumps[7].Linear.rActualTorque;
GVL_HMI.stIOTerm29.bAxisHomed[1] 		:= GVL_Motion.aPumps[7].Linear.iHomed;
GVL_HMI.stIOTerm29.bAxisError[1] 		:= GVL_Motion.aPumps[7].Linear.iError;
GVL_HMI.stIOTerm29.nErrorCode[1] 		:= GVL_Motion.aPumps[7].Linear.nErrorCode;
GVL_HMI.stIOTerm29.bAxisOperational[2] 	:= GVL_Motion.aPumps[7].Rotary.iOperational;
GVL_HMI.stIOTerm29.rActualPosition[2] 	:= GVL_Motion.aPumps[7].Rotary.rActualPos;
GVL_HMI.stIOTerm29.rActualVelocity[2] 	:= GVL_Motion.aPumps[7].Rotary.rActualVel;
GVL_HMI.stIOTerm29.rActualTorque[2] 	:= GVL_Motion.aPumps[7].Rotary.rActualTorque;
GVL_HMI.stIOTerm29.bAxisHomed[2] 		:= GVL_Motion.aPumps[7].Rotary.iHomed;
GVL_HMI.stIOTerm29.bAxisError[2] 		:= GVL_Motion.aPumps[7].Rotary.iError;
GVL_HMI.stIOTerm29.nErrorCode[2] 		:= GVL_Motion.aPumps[7].Rotary.nErrorCode;

(* <EL7062 Terminal 30> -------------------------------------------------------------------------------------------------------------*)
GVL_HMI.stIOTerm30.bAxisOperational[1] 	:= GVL_Motion.aPumps[8].Linear.iOperational;
GVL_HMI.stIOTerm30.rActualPosition[1] 	:= GVL_Motion.aPumps[8].Linear.rActualPos;
GVL_HMI.stIOTerm30.rActualVelocity[1] 	:= GVL_Motion.aPumps[8].Linear.rActualVel;
GVL_HMI.stIOTerm30.rActualTorque[1] 	:= GVL_Motion.aPumps[8].Linear.rActualTorque;
GVL_HMI.stIOTerm30.bAxisHomed[1] 		:= GVL_Motion.aPumps[8].Linear.iHomed;
GVL_HMI.stIOTerm30.bAxisError[1] 		:= GVL_Motion.aPumps[8].Linear.iError;
GVL_HMI.stIOTerm30.nErrorCode[1] 		:= GVL_Motion.aPumps[8].Linear.nErrorCode;
GVL_HMI.stIOTerm30.bAxisOperational[2] 	:= GVL_Motion.aPumps[8].Rotary.iOperational;
GVL_HMI.stIOTerm30.rActualPosition[2] 	:= GVL_Motion.aPumps[8].Rotary.rActualPos;
GVL_HMI.stIOTerm30.rActualVelocity[2] 	:= GVL_Motion.aPumps[8].Rotary.rActualVel;
GVL_HMI.stIOTerm30.rActualTorque[2] 	:= GVL_Motion.aPumps[8].Rotary.rActualTorque;
GVL_HMI.stIOTerm30.bAxisHomed[2] 		:= GVL_Motion.aPumps[8].Rotary.iHomed;
GVL_HMI.stIOTerm30.bAxisError[2] 		:= GVL_Motion.aPumps[8].Rotary.iError;
GVL_HMI.stIOTerm30.nErrorCode[2] 		:= GVL_Motion.aPumps[8].Rotary.nErrorCode;

(* <EL7062 Terminal 31> -------------------------------------------------------------------------------------------------------------*)
GVL_HMI.stIOTerm31.bAxisOperational[1] 	:= GVL_Motion.aPumps[9].Linear.iOperational;
GVL_HMI.stIOTerm31.rActualPosition[1] 	:= GVL_Motion.aPumps[9].Linear.rActualPos;
GVL_HMI.stIOTerm31.rActualVelocity[1] 	:= GVL_Motion.aPumps[9].Linear.rActualVel;
GVL_HMI.stIOTerm31.rActualTorque[1] 	:= GVL_Motion.aPumps[9].Linear.rActualTorque;
GVL_HMI.stIOTerm31.bAxisHomed[1] 		:= GVL_Motion.aPumps[9].Linear.iHomed;
GVL_HMI.stIOTerm31.bAxisError[1] 		:= GVL_Motion.aPumps[9].Linear.iError;
GVL_HMI.stIOTerm31.nErrorCode[1] 		:= GVL_Motion.aPumps[9].Linear.nErrorCode;
GVL_HMI.stIOTerm31.bAxisOperational[2] 	:= GVL_Motion.aPumps[9].Rotary.iOperational;
GVL_HMI.stIOTerm31.rActualPosition[2] 	:= GVL_Motion.aPumps[9].Rotary.rActualPos;
GVL_HMI.stIOTerm31.rActualVelocity[2] 	:= GVL_Motion.aPumps[9].Rotary.rActualVel;
GVL_HMI.stIOTerm31.rActualTorque[2] 	:= GVL_Motion.aPumps[9].Rotary.rActualTorque;
GVL_HMI.stIOTerm31.bAxisHomed[2] 		:= GVL_Motion.aPumps[9].Rotary.iHomed;
GVL_HMI.stIOTerm31.bAxisError[2] 		:= GVL_Motion.aPumps[9].Rotary.iError;
GVL_HMI.stIOTerm31.nErrorCode[2] 		:= GVL_Motion.aPumps[9].Rotary.nErrorCode;

(* <EL7062 Terminal 32> -------------------------------------------------------------------------------------------------------------*)
GVL_HMI.stIOTerm32.bAxisOperational[1] 	:= GVL_Motion.aPumps[10].Linear.iOperational;
GVL_HMI.stIOTerm32.rActualPosition[1] 	:= GVL_Motion.aPumps[10].Linear.rActualPos;
GVL_HMI.stIOTerm32.rActualVelocity[1] 	:= GVL_Motion.aPumps[10].Linear.rActualVel;
GVL_HMI.stIOTerm32.rActualTorque[1] 	:= GVL_Motion.aPumps[10].Linear.rActualTorque;
GVL_HMI.stIOTerm32.bAxisHomed[1] 		:= GVL_Motion.aPumps[10].Linear.iHomed;
GVL_HMI.stIOTerm32.bAxisError[1] 		:= GVL_Motion.aPumps[10].Linear.iError;
GVL_HMI.stIOTerm32.nErrorCode[1] 		:= GVL_Motion.aPumps[10].Linear.nErrorCode;
GVL_HMI.stIOTerm32.bAxisOperational[2] 	:= GVL_Motion.aPumps[10].Rotary.iOperational;
GVL_HMI.stIOTerm32.rActualPosition[2] 	:= GVL_Motion.aPumps[10].Rotary.rActualPos;
GVL_HMI.stIOTerm32.rActualVelocity[2] 	:= GVL_Motion.aPumps[10].Rotary.rActualVel;
GVL_HMI.stIOTerm32.rActualTorque[2] 	:= GVL_Motion.aPumps[10].Rotary.rActualTorque;
GVL_HMI.stIOTerm32.bAxisHomed[2] 		:= GVL_Motion.aPumps[10].Rotary.iHomed;
GVL_HMI.stIOTerm32.bAxisError[2] 		:= GVL_Motion.aPumps[10].Rotary.iError;
GVL_HMI.stIOTerm32.nErrorCode[2] 		:= GVL_Motion.aPumps[10].Rotary.nErrorCode;

(* <EL7062 Terminal 34> -------------------------------------------------------------------------------------------------------------*)
GVL_HMI.stIOTerm34.bAxisOperational 	:= GVL_Motion.M1Motor.iOperational;
GVL_HMI.stIOTerm34.bAxisHomed 			:= GVL_Motion.M1Motor.iHomed;
GVL_HMI.stIOTerm34.bNotMoving			:= GVL_Motion.M1Motor.iNotMoving;
GVL_HMI.stIOTerm34.bAxisError 			:= GVL_Motion.M1Motor.iError;
GVL_HMI.stIOTerm34.bDriveError 			:= GVL_Motion.M1Motor.iError;
GVL_HMI.stIOTerm34.nErrorCode 			:= GVL_Motion.M1Motor.nErrorCode;
GVL_HMI.stIOTerm34.rActualPosition 		:= LINT_TO_LREAL(TRUNC(GVL_Motion.M1Motor.rActualPos * 1000)) /1000;
GVL_HMI.stIOTerm34.rActualVelocity 		:= LINT_TO_LREAL(TRUNC(GVL_Motion.M1Motor.rActualVel * 1000)) /1000;

(* <Box 1 ifm AL1333> --------------------------------------------------------------------------------------------------------------*)
GVL_HMI.aIOBox1[1] := GVL_HMI.HMIAnimation.aSolventLevel[1];
GVL_HMI.aIOBox1[2] := GVL_HMI.HMIAnimation.aSolventLevel[2];
GVL_HMI.aIOBox1[3] := GVL_HMI.HMIAnimation.aSolventLevel[3];
GVL_HMI.aIOBox1[4] := GVL_HMI.HMIAnimation.aSolventLevel[4];
GVL_HMI.aIOBox1[5] := GVL_HMI.HMIAnimation.rWasteLevel;

(* <Box 2 AMI8000 - Valve 1> -------------------------------------------------------------------------------------------------------------*)
GVL_HMI.aIOAMI8000[1].bAxisOperational 	:= GVL_Motion.aValves[1].iOperational;
GVL_HMI.aIOAMI8000[1].bAxisHomed 		:= GVL_Motion.aValves[1].iHomed;
GVL_HMI.aIOAMI8000[1].bNotMoving 		:= GVL_Motion.aValves[1].iNotMoving;
GVL_HMI.aIOAMI8000[1].bAxisError 		:= GVL_Motion.aValves[1].iError;
GVL_HMI.aIOAMI8000[1].nErrorCode 		:= GVL_Motion.aValves[1].nErrorCode;
GVL_HMI.aIOAMI8000[1].rActualPosition 	:= LINT_TO_LREAL(TRUNC(GVL_Motion.aValves[1].rActualPos* 1000)) /1000;
GVL_HMI.aIOAMI8000[1].rActualVelocity 	:= LINT_TO_LREAL(TRUNC(GVL_Motion.aValves[1].rActualVel* 1000)) /1000;

(* <Box 3 AMI8000 - Valve 2> -------------------------------------------------------------------------------------------------------------*)
GVL_HMI.aIOAMI8000[2].bAxisOperational 	:= GVL_Motion.aValves[2].iOperational;
GVL_HMI.aIOAMI8000[2].bAxisHomed 		:= GVL_Motion.aValves[2].iHomed;
GVL_HMI.aIOAMI8000[2].bNotMoving 		:= GVL_Motion.aValves[2].iNotMoving;
GVL_HMI.aIOAMI8000[2].bAxisError 		:= GVL_Motion.aValves[2].iError;
GVL_HMI.aIOAMI8000[2].nErrorCode 		:= GVL_Motion.aValves[2].nErrorCode;
GVL_HMI.aIOAMI8000[2].rActualPosition 	:= LINT_TO_LREAL(TRUNC(GVL_Motion.aValves[2].rActualPos* 1000)) /1000;
GVL_HMI.aIOAMI8000[2].rActualVelocity 	:= LINT_TO_LREAL(TRUNC(GVL_Motion.aValves[2].rActualVel* 1000)) /1000;

(* <Box 4 AMI8000 - Valve 3> -------------------------------------------------------------------------------------------------------------*)
GVL_HMI.aIOAMI8000[3].bAxisOperational 	:= GVL_Motion.aValves[3].iOperational;
GVL_HMI.aIOAMI8000[3].bAxisHomed 		:= GVL_Motion.aValves[3].iHomed;
GVL_HMI.aIOAMI8000[3].bNotMoving 		:= GVL_Motion.aValves[3].iNotMoving;
GVL_HMI.aIOAMI8000[3].bAxisError 		:= GVL_Motion.aValves[3].iError;
GVL_HMI.aIOAMI8000[3].nErrorCode 		:= GVL_Motion.aValves[3].nErrorCode;
GVL_HMI.aIOAMI8000[3].rActualPosition 	:= LINT_TO_LREAL(TRUNC(GVL_Motion.aValves[3].rActualPos* 1000)) /1000;
GVL_HMI.aIOAMI8000[3].rActualVelocity 	:= LINT_TO_LREAL(TRUNC(GVL_Motion.aValves[3].rActualVel* 1000)) /1000;

(* <Box 5 AMI8000 - Valve 4> -------------------------------------------------------------------------------------------------------------*)
GVL_HMI.aIOAMI8000[4].bAxisOperational 	:= GVL_Motion.aValves[4].iOperational;
GVL_HMI.aIOAMI8000[4].bAxisHomed 		:= GVL_Motion.aValves[4].iHomed;
GVL_HMI.aIOAMI8000[4].bNotMoving 		:= GVL_Motion.aValves[4].iNotMoving;
GVL_HMI.aIOAMI8000[4].bAxisError 		:= GVL_Motion.aValves[4].iError;
GVL_HMI.aIOAMI8000[4].nErrorCode 		:= GVL_Motion.aValves[4].nErrorCode;
GVL_HMI.aIOAMI8000[4].rActualPosition 	:= LINT_TO_LREAL(TRUNC(GVL_Motion.aValves[4].rActualPos* 1000)) /1000;
GVL_HMI.aIOAMI8000[4].rActualVelocity 	:= LINT_TO_LREAL(TRUNC(GVL_Motion.aValves[4].rActualVel* 1000)) /1000;

(* <Box 6 AMI8000 - Valve 5> -------------------------------------------------------------------------------------------------------------*)
GVL_HMI.aIOAMI8000[5].bAxisOperational 	:= GVL_Motion.aValves[5].iOperational;
GVL_HMI.aIOAMI8000[5].bAxisHomed 		:= GVL_Motion.aValves[5].iHomed;
GVL_HMI.aIOAMI8000[5].bNotMoving 		:= GVL_Motion.aValves[5].iNotMoving;
GVL_HMI.aIOAMI8000[5].bAxisError 		:= GVL_Motion.aValves[5].iError;
GVL_HMI.aIOAMI8000[5].nErrorCode 		:= GVL_Motion.aValves[5].nErrorCode;
GVL_HMI.aIOAMI8000[5].rActualPosition 	:= LINT_TO_LREAL(TRUNC(GVL_Motion.aValves[5].rActualPos* 1000)) /1000;
GVL_HMI.aIOAMI8000[5].rActualVelocity 	:= LINT_TO_LREAL(TRUNC(GVL_Motion.aValves[5].rActualVel* 1000)) /1000;

(* <Motors nState> -----------------------------------------------------------------------------------------------------------------*)
GVL_IO.nAX8108T34State := GVL_Motion.M1Motor.nState; //M1
GVL_IO.nEL7211T15State := GVL_Motion.M2Motor.nState; //M2
GVL_IO.nEL7211T16State := GVL_Motion.M3Motor.nState; //M3
GVL_IO.nAMI8000Box8State := GVL_Motion.aValves[1].nState; //Valve 1
GVL_IO.nAMI8000Box9State := GVL_Motion.aValves[2].nState; //Valve 2
GVL_IO.nAMI8000Box10State := GVL_Motion.aValves[3].nState; //Valve 3
GVL_IO.nAMI8000Box11State := GVL_Motion.aValves[4].nState; //Valve 4
GVL_IO.nAMI8000Box12State := GVL_Motion.aValves[5].nState; //Valve 5
GVL_IO.nEL7062T23State := GVL_Motion.aPumps[1].Linear.nState; //Pump1 Terminal
GVL_IO.nEL7062T24State := GVL_Motion.aPumps[2].Linear.nState; //Pump2 Terminal
GVL_IO.nEL7062T25State := GVL_Motion.aPumps[3].Linear.nState; //Pump3 Terminal
GVL_IO.nEL7062T26State := GVL_Motion.aPumps[4].Linear.nState; //Pump4 Terminal
GVL_IO.nEL7062T27State := GVL_Motion.aPumps[5].Linear.nState; //Pump5 Terminal
GVL_IO.nEL7062T28State := GVL_Motion.aPumps[6].Linear.nState; //Pump6 Terminal
GVL_IO.nEL7062T29State := GVL_Motion.aPumps[7].Linear.nState; //Pump7 Terminal
GVL_IO.nEL7062T30State := GVL_Motion.aPumps[8].Linear.nState; //Pump8 Terminal
GVL_IO.nEL7062T31State := GVL_Motion.aPumps[9].Linear.nState; //Pump9 Terminal
GVL_IO.nEL7062T32State := GVL_Motion.aPumps[10].Linear.nState; //Pump10 Terminal
END_ACTION

ACTION ACT_JarsAnimation:
(* Jar Animation *)

//when pumping into jars? Pump positive movement  

FOR i := 1 TO cJarsCount DO

    // ----------------- 1) Leitura posição (em VOLTAS) ------------------------
    curTurns := GVL_Motion.aPumps[i].Rotary.Axis.NcToPlc.ActPos / aUnitsPerTurn[i];

    // 2) Primeira amostra: inicializa e publica
    IF NOT aPrevInit[i] THEN
        aPrevTurns[i]     := curTurns;
        aPrevInit[i]      := TRUE;
        aDispMl[i]        := aJarMl[i];      // alinhar disp ao interno
        GVL_HMI.HmiAnimation.rJarFillAnimation[i] :=
            LIMIT(0.0, (aDispMl[i] / cJarCapacity_ml) * 100.0, 100.0);
        CONTINUE;
    END_IF

    // ----------------- 3) Delta e direção ------------------------------------
    deltaTurns := curTurns - aPrevTurns[i];
    dMl := deltaTurns * GVL_Motion.aPumps[i].Rotary.rPumpFactorFillJars;

    dir := 0;
    IF GVL_Motion.aPumps[i].Rotary.bPositiveDirection THEN
        dir := 1;
    ELSIF GVL_Motion.aPumps[i].Rotary.bNegativeDirection THEN
        dir := -1;
    ELSE
        IF dMl >  0.0 THEN dir := 1; END_IF
        IF dMl <  0.0 THEN dir := -1; END_IF
    END_IF

    // Sem movimento relevante?
    IF (ABS(deltaTurns) <= cEpsTurns) OR (dir = 0) THEN
        // publica (considerando se estava/está em recirculação)
        valIdx := ((i + 1) / 2); // 1&2->1, 3&4->2, ..., 9&10->5
        bRecircActive := (valIdx >= 1) AND (valIdx <= 5) AND
                         (GVL_Motion.aValves[valIdx].rActualPos >= cRecircLowDeg) AND
                         (GVL_Motion.aValves[valIdx].rActualPos <= cRecircHighDeg);

        IF bRecircActive THEN
            // sem movimento, mantém exibição atual (aDispMl)
        ELSE
            // fora da recirculação, exibe o interno
            aDispMl[i] := aJarMl[i];
        END_IF

        GVL_HMI.HmiAnimation.rJarFillAnimation[i] :=
            LIMIT(0.0, (aDispMl[i] / cJarCapacity_ml) * 100.0, 100.0);
        aPrevTurns[i] := curTurns;
        aRecircWasActive[i] := bRecircActive;
        CONTINUE;
    END_IF

    // ----------------- 4) Checar recirculação --------------------------------
    valIdx := ((i + 1) / 2);
    bRecircActive := (valIdx >= 1) AND (valIdx <= 5) AND
                     (GVL_Motion.aValves[valIdx].rActualPos >= cRecircLowDeg) AND
                     (GVL_Motion.aValves[valIdx].rActualPos <= cRecircHighDeg);

    IF bRecircActive THEN
        // Entrando agora? salva patamar base e sincroniza display
        IF NOT aRecircWasActive[i] THEN
            aRecircBaseMl[i] := aJarMl[i];     // patamar que “voltará” quando positivo
            aDispMl[i]       := aJarMl[i];     // start visual no nível atual
        END_IF

        // Anda a exibição “na razão da bomba”, sem alterar aJarMl
        IF dir < 0 THEN
            // cair até 20 mL gradualmente
            aDispMl[i] := MAX(cRecircDisplayMin_ml, aDispMl[i] - ABS(dMl));
        ELSIF dir > 0 THEN
            // subir de volta ao patamar base
            aDispMl[i] := MIN(aRecircBaseMl[i], aDispMl[i] + ABS(dMl));
        END_IF

        // Publicar exibição
        GVL_HMI.HmiAnimation.rJarFillAnimation[i] :=
            LIMIT(0.0, (aDispMl[i] / cJarCapacity_ml) * 100.0, 100.0);

        // Atualizações de referência e flags
        aPrevTurns[i]      := curTurns;
        aRecircWasActive[i]:= TRUE;

        // Pula integração/DeadVol: jar interno não muda em recirculação
        CONTINUE;
    END_IF

    // Saiu de recirculação agora? ressincroniza exibição com interno
    IF aRecircWasActive[i] AND (NOT bRecircActive) THEN
        aDispMl[i] := aJarMl[i];
    END_IF
    aRecircWasActive[i] := FALSE;

    // ----------------- 5) Lógica normal (fora da recirculação) ---------------
    // Mudou direção? novo segmento
    IF aSegDir[i] <> dir THEN
        aSegDir[i]       := dir;
        aSegAbsMl[i]     := 0.0;
        aSegAbsMlPrev[i] := 0.0;
    END_IF

    // Acumula módulo de mL neste segmento
    aSegAbsMlPrev[i] := aSegAbsMl[i];
    aSegAbsMl[i]     := aSegAbsMl[i] + ABS(dMl);

    // Aplica DeadVol por segmento:
    //  + Encher: só após exceder DeadVol o jar sobe
    //  - Esvaziar: só até (seg - DeadVol) o jar desce (últimos DeadVol não mexem)
    effDeltaMl := 0.0;

    IF dir = 1 THEN
        segNowEff  := MAX(0.0, aSegAbsMl[i]     - aDeadVolCfg_ml[i]);
        segPrevEff := MAX(0.0, aSegAbsMlPrev[i] - aDeadVolCfg_ml[i]);
        effDeltaMl := segNowEff - segPrevEff;        // aumenta jar
        aJarMl[i]  := aJarMl[i] + effDeltaMl;

    ELSIF dir = -1 THEN
        segNowEff  := MAX(0.0, aSegAbsMl[i]     - aDeadVolCfg_ml[i]);
        segPrevEff := MAX(0.0, aSegAbsMlPrev[i] - aDeadVolCfg_ml[i]);
        effDeltaMl := segNowEff - segPrevEff;        // diminui jar
        aJarMl[i]  := aJarMl[i] - effDeltaMl;
    END_IF

    // Limites físicos
    IF aJarMl[i] < 0.0 THEN aJarMl[i] := 0.0; END_IF
    IF aJarMl[i] > cJarCapacity_ml THEN aJarMl[i] := cJarCapacity_ml; END_IF

    // Publica (fora da recirculação, exibe o interno)
    aDispMl[i] := aJarMl[i];
    GVL_HMI.HmiAnimation.rJarFillAnimation[i] :=
        LIMIT(0.0, (aDispMl[i] / cJarCapacity_ml) * 100.0, 100.0);

    // Referência
    aPrevTurns[i] := curTurns;

END_FOR;
END_ACTION

ACTION ACT_M1Animation:
//M1 Motor vertical Axis Animation
IF GVL_Motion.bInitialHomingDone THEN
	// Read the end of scale value
	cM1MaxPosition := GVL_Settings.stMachineParam.aM1Position[2];	

	// Read motor Position
	rM1MotorPosition := GVL_Motion.M1Motor.rActualPos;
	
	//Check if cM1MaxPosition has a number different from 0
	IF cM1MaxPosition < 0 THEN
		// Scaling the motor position (0 = 0%, -320 = 100%)
		rM1MotorPositionPerc := ((rM1MotorPosition - cM1MinPosition) / (cM1MaxPosition - cM1MinPosition)) * 100.0; //Error 06/10/25
	ELSE
		rM1MotorPositionPerc := 0;
	END_IF
	
	// Limits value in the range 0 and 100%
	IF rM1MotorPositionPerc < 0 THEN
		rM1MotorPositionPerc := 0;
	ELSIF rM1MotorPositionPerc > 100 THEN
		rM1MotorPositionPerc := 100;
	END_IF
	
	GVL_HMI.HMIAnimation.rM1VerticalAnimation := 0 + (TO_REAL(rM1MotorPositionPerc)*1.55); //Adding y pixel home and sending the scaled value throug GVL_HMI
ELSE
	GVL_HMI.HMIAnimation.rM1VerticalAnimation := 0; //Default Value
END_IF
END_ACTION

ACTION ACT_M2Animation:
//M2 HMI object moves from pixel 455 (0 Position) up to 555 (Max position = -170mm)
//M2 Motor vertical Axis Animation
IF GVL_Motion.bInitialHomingDone THEN
	// Read the end of scale value
	cM2MaxPosition := GVL_Settings.stMachineParam.aM2Position[4]; //Calibration Position witch is the most away position the motor will reach	

	// Read motor Position
	rM2MotorPosition := GVL_Motion.M2Motor.rActualPos;
	
	//Check if cM2MaxPosition has a number different from 0
	IF cM2MaxPosition < 0 THEN
		// Scaling the motor position (0 = 0%, -320 = 100%)
		rM2MotorPositionPerc := ((rM2MotorPosition - cM2MinPosition) / (cM2MaxPosition - cM2MinPosition)) * 100.0; //Error 06/10/25
	ELSE
		rM2MotorPositionPerc := 0;
	END_IF
	
	// Limits value in the range 0 and 100%
	IF rM2MotorPositionPerc < 0 THEN
		rM2MotorPositionPerc := 0;
	ELSIF rM2MotorPositionPerc > 100 THEN
		rM2MotorPositionPerc := 100;
	END_IF
	
	GVL_HMI.HMIAnimation.rM2VerticalAnimation := 0 + (TO_REAL(rM2MotorPositionPerc)*0.9); //Adding y pixel home and sending the scaled value throug GVL_HMI
ELSE
	GVL_HMI.HMIAnimation.rM2VerticalAnimation := 0; //Default Value
END_IF
END_ACTION

END_PROGRAM

(* stored: Version 1.1.0.1, ProductVersion 3.1.4024.15
   POU PRG_HMIControl: Id {978beb02-d146-472c-ad6b-2f8739fa70ac}, SpecialFunc None
   Action ACT_CalibrationArrows: Id {79e47b94-61cf-47c5-8acf-43afca6d34ed}
   Action ACT_IOControls: Id {9ed40c73-f032-4eec-b4aa-fa2f87be3486}
   Action ACT_JarsAnimation: Id {15390b10-db75-4567-a585-5216d7eaf80d}
   Action ACT_M1Animation: Id {5ca7e550-b195-4047-b743-192dee895467}
   Action ACT_M2Animation: Id {2010a8e8-186b-452d-a6f4-adbd9f915f7d} *)
